(*********************************** G.D S.p.A. - Technical Department ***********************************
============= PROGRAM INFO ============
FOLDER:             TBD
MACHINES INVOLVED:  TBD 

============= DESCRIPTION =============
Machine notaus series

============= REVISIONS ===============
Date		Version	 	Author      	Description             
----------	-------		------------  	--------------------------------------------
2020/02/10 	0000.00	 	M.Grasso		Creation of the PRG

**********************************************************************************************************)
(*$R process_ref:= prc; $*)

PROGRAM csp_main_safety_emergency
VAR
	prc:											process;
	prc_path:										STRING;
	
 END_VAR

_read_var_input();

_objects_manager();

IF NOT objects_running()
THEN
	RETURN;	
END_IF

_read_process_image();

_mode_manager();

CASE process_get_mode(prc) OF
	MODE_ABSENT,
	MODE_INACTIVE:
		RETURN;
	MODE_TEST:
		;
END_CASE

_set_runtime_properties();

(********************************* BODY *********************************)
IF	descriptor_get_reset_edge(prc.descriptor)
THEN
	safety_integrated_series_close(sis);
	safety_integrated_series_close(delayed_sis);
END_IF
(************************************************************************)

_handle_messages();

_write_output();

ACTION _handle_messages:
;
END_ACTION

ACTION _handle_process_test:
;
END_ACTION

ACTION _mode_manager:
IF process_mode_req_is_pending(prc)
THEN
    process_apply_mode_req_first_step(prc);
    CASE process_get_mode(prc) OF
        MODE_TO_ABSENT:
			;
        MODE_TO_INACTIVE:
			;
        MODE_TO_TEST:
			;
        MODE_TO_OPERATIONAL:
			;
    END_CASE
    process_apply_mode_req_second_step(prc);
END_IF
END_ACTION

ACTION _objects_manager:
IF objects_initialization()
THEN

	sub_process_init(
		object_name								:= 'csp_main_safety_emergency.prc', 
		process									:= csp_main_safety.prc, 
		CONVERSION_this							:= prc);
		
	prc_path 									:= process_get_path(prc);

END_IF


IF	objects_running()
THEN
    process_cycle(prc);
END_IF
END_ACTION

ACTION _read_process_image:
;
END_ACTION

ACTION _read_var_input:
;
END_ACTION

ACTION _set_runtime_properties:
;
END_ACTION

ACTION _write_output:
;
END_ACTION

END_PROGRAM

(* stored: Version 1.1.0.1, ProductVersion 3.1.4022.12
   POU csp_main_safety_emergency: Id {e63aabb5-2a78-4e76-8155-f1861e9255e6}, SpecialFunc None
   Action _handle_messages: Id {5c007f66-8f63-4985-a15b-0d1876b3e2d2}
   Action _handle_process_test: Id {e11b9bcc-ab98-44d5-a917-4f7b3463a414}
   Action _mode_manager: Id {a61ff840-98e9-45a7-a221-a22fb9b1fd3e}
   Action _objects_manager: Id {23bcd131-068d-4171-8fbb-0098a13cd2b2}
   Action _read_process_image: Id {99063b59-d0eb-41b9-a81f-b2521de74fe9}
   Action _read_var_input: Id {cec48ea1-d828-4be1-b479-df1dd78eb74f}
   Action _set_runtime_properties: Id {4e3d030b-4bda-4fd0-b21c-fab250f47b24}
   Action _write_output: Id {9743563d-c403-4122-9120-b8a1aa215db3} *)
